PROGRAM Trips
VAR
	bTest							: BOOL;
	//delay2s : Delay2s;
	evtLogger						: FB_TcEventLogger;
	
	ACintLockRlyFaultDelay_PT		: TIME := T#2S;
	DumpRlyFaultDelay_PT			: TIME := T#2S;
	//DumpRly2FaultDelay_PT			: TIME := T#2S;
	ChrgRlyFaultDelay_PT			: TIME := T#1S;
	
	i : INT := 1;  //charger 1-8
	j : INT := 1; //section 1-3
	k : INT := 1; //section 1-4, might not need 
END_VAR


//MCP Input Trips
IF MCP_IO.MasterStopPB_Pressed = TRUE THEN
	Trips_DB.MasterStopPBPressed := TRUE;	
END_IF;

IF MCP_IO.CageEstopCircuitOK = FALSE THEN
	Trips_DB.CaseEStopCircuitBroken := TRUE; 
END_IF;

IF MCP_IO.AutoModeSelected = FALSE THEN
	Trips_DB.ManualModeSelected := TRUE; //may not be a trip
	ELSE
		Trips_DB.ManualModeSelected := FALSE;
END_IF;

IF MCP_IO.PSU1_DCOK = FALSE THEN
	Trips_DB.MCPLossDCpower := TRUE; 
END_IF;

// mapping pnumatic and dc power to trips
FOR k := 1 TO 4 BY 1 DO
	Trips_DB.Section[k].LossPneumaticPressure := LCP.Section[k].LossPneumaticPressure;
	Trips_DB.Section[k].LossDCPower := NOT LCP.Section[k].PSU1_DCOK;
END_FOR;


//any charge relay fail
IF Trips_DB.Section[1].Peak.ChargeRelay1_Failed = TRUE OR
	Trips_DB.Section[1].Peak.ChargeRelay2_Failed = TRUE OR
	Trips_DB.Section[1].Sust.ChargeRelay1_Failed = TRUE OR
	Trips_DB.Section[1].Sust.ChargeRelay2_Failed = TRUE OR
	Trips_DB.Section[2].Peak.ChargeRelay1_Failed = TRUE OR
	Trips_DB.Section[2].Peak.ChargeRelay2_Failed = TRUE OR
	Trips_DB.Section[2].Sust.ChargeRelay1_Failed = TRUE OR
	Trips_DB.Section[2].Sust.ChargeRelay2_Failed = TRUE OR
	Trips_DB.Section[3].Peak.ChargeRelay1_Failed = TRUE OR
	Trips_DB.Section[3].Peak.ChargeRelay2_Failed = TRUE OR
	Trips_DB.Section[3].Sust.ChargeRelay1_Failed = TRUE OR
	Trips_DB.Section[3].Sust.ChargeRelay2_Failed = TRUE OR
	Trips_DB.Section[4].Form.ChargeRelay1_Failed = TRUE OR 
	Trips_DB.Section[4].Form.ChargeRelay2_Failed = TRUE OR 
	Trips_DB.Section[4].Form.PreFormChrgRlyFailed = TRUE OR 
	Trips_DB.Section[4].Form.FormTrigChrgRlyFailed = TRUE OR
	Trips_DB.Section[4].Form.PreFormTrigChrgRlyFailed = TRUE		
	THEN 
		Trips_DB.AnyChargeRlyFail := TRUE;
	ELSE
		Trips_DB.AnyChargeRlyFail := FALSE;
END_IF;

//any dump relay fail
IF Trips_DB.Section[1].Peak.DumpRelay1_Failed = TRUE OR
	Trips_DB.Section[1].Peak.DumpRelay2_Failed = TRUE OR
	Trips_DB.Section[1].Sust.DumpRelay1_Failed = TRUE OR
	Trips_DB.Section[1].Sust.DumpRelay2_Failed = TRUE OR
	Trips_DB.Section[2].Peak.DumpRelay1_Failed = TRUE OR
	Trips_DB.Section[2].Peak.DumpRelay2_Failed = TRUE OR
	Trips_DB.Section[2].Sust.DumpRelay1_Failed = TRUE OR
	Trips_DB.Section[2].Sust.DumpRelay2_Failed = TRUE OR
	Trips_DB.Section[3].Peak.DumpRelay1_Failed = TRUE OR
	Trips_DB.Section[3].Peak.DumpRelay2_Failed = TRUE OR
	Trips_DB.Section[3].Sust.DumpRelay1_Failed = TRUE OR
	Trips_DB.Section[3].Sust.DumpRelay2_Failed = TRUE OR
	Trips_DB.Section[4].Form.DumpRelay1_Failed = TRUE OR 
	Trips_DB.Section[4].Form.DumpRelay2_Failed = TRUE OR 
	Trips_DB.Section[4].Form.PreFormDumpRlyFailed = TRUE OR 
	Trips_DB.Section[4].Form.FormTrigDumpRly1Failed = TRUE OR
	Trips_DB.Section[4].Form.PreFormTrigDumpRly1Failed = TRUE		
	THEN 
		Trips_DB.AnyDumpRlyFail := TRUE;
	ELSE
		Trips_DB.AnyDumpRlyFail := FALSE;
END_IF;

//if relays failed, chargers faulted, loss pneumatic pressure, or loss dc power then 
//Trips_DB.Section[j].SystemTripped := TRUE;

//system trip 
//section 1-3
FOR j := 1 TO 3 BY 1 DO
	IF Trips_DB.Section[j].LossDCPower = TRUE OR 
		Trips_DB.Section[j].LossPneumaticPressure = TRUE OR
		Trips_DB.Section[j].Peak.ChargeRelay1_Failed = TRUE OR
		Trips_DB.Section[j].Peak.ChargeRelay2_Failed = TRUE OR
		Trips_DB.Section[j].Peak.DumpRelay1_Failed = TRUE OR
		Trips_DB.Section[j].Peak.DumpRelay2_Failed = TRUE OR
		Trips_DB.Section[j].Sust.ChargeRelay1_Failed = TRUE OR
		Trips_DB.Section[j].Sust.ChargeRelay2_Failed = TRUE OR
		Trips_DB.Section[j].Sust.DumpRelay1_Failed = TRUE OR
		Trips_DB.Section[j].Sust.DumpRelay2_Failed = TRUE 
		// shorted when not supposed to ?
		THEN
			Trips_DB.Section[j].SystemTripped := TRUE;
	END_IF;
END_FOR;

//formation
IF Trips_DB.Section[4].LossDCPower = TRUE OR 
	Trips_DB.Section[4].LossPneumaticPressure = TRUE OR
	Trips_DB.Section[4].Form.ChargeRelay1_Failed = TRUE OR
	Trips_DB.Section[4].Form.ChargeRelay2_Failed = TRUE OR
	Trips_DB.Section[4].Form.DumpRelay1_Failed = TRUE OR
	Trips_DB.Section[4].Form.DumpRelay2_Failed = TRUE OR
	Trips_DB.Section[4].Form.PreFormChrgRlyFailed = TRUE OR
	Trips_DB.Section[4].Form.FormTrigChrgRlyFailed = TRUE OR
	Trips_DB.Section[4].Form.PreFormTrigChrgRlyFailed = TRUE OR
	Trips_DB.Section[4].Form.PreFormDumpRlyFailed = TRUE OR
	Trips_DB.Section[4].Form.FormTrigDumpRly1Failed = TRUE OR
	Trips_DB.Section[4].Form.PreFormTrigDumpRly1Failed = TRUE
	THEN
		Trips_DB.Section[4].SystemTripped := TRUE;
END_IF;


//Charger faults
FOR i := 1 TO 8 BY 1 DO
	//OVERTEMP 
	IF MCP_IO.Charger[i].OverTemp = TRUE THEN
		Trips_DB.AnyChargerOverTemp := TRUE;  
	END_IF;
	//Load faults
	IF MCP_IO.Charger[i].LoadFaulted = TRUE THEN
		Trips_DB.AnyChargerLoadFault := TRUE;  
	END_IF;
	//Interlock Open
	IF MCP_IO.Charger[i].InterlockOpen = TRUE THEN
		Trips_DB.AnyChargerInterlockOpen := TRUE;  
	END_IF;
	
END_FOR;

//Charger summary faults
FOR i := 1 TO 8 BY 1 DO
	IF MCP_IO.Charger[i].SummaryFaulted = TRUE THEN
		Trips_DB.AnyChargerFaulted := TRUE;  
	END_IF;
END_FOR;

//MCP trip
IF Trips_DB.AnyChargerFaulted = TRUE OR 
	Trips_DB.MasterStopPBPressed = TRUE OR
	Trips_DB.CaseEStopCircuitBroken = TRUE OR
	Trips_DB.MCPLossDCpower = TRUE 
	THEN
		Trips_DB.MCPsystemTripped := TRUE;
END_IF


//*******************E-Stop Trips
IF MCP_IO.MasterStopPB_Pressed = TRUE OR MCP_IO.CageEstopCircuitOK THEN
	Trips_DB.AnyEstopPressed := TRUE;  
END_IF;	

//*********************DC PSU
IF MCP_IO.PSU1_DCOK = TRUE AND 
	LCP.Section[1].PSU1_DCOK = TRUE AND
	LCP.Section[2].PSU1_DCOK = TRUE AND
	LCP.Section[3].PSU1_DCOK = TRUE AND
	LCP.Section[4].PSU1_DCOK = TRUE 
	THEN
		TRIPS_DB.AllDCpsuOK := TRUE;
	ELSE 
		TRIPS_DB.AllDCpsuOK := FALSE;
END_IF;

//Relay faults***************************************
//section 1 - 3
FOR j := 1 TO 3 BY 1 DO
	//Peak Charge rly1
		//fail to close
	IF LCP.Section[j].Peak.CloseChargeRelay1 = TRUE AND LCP.Section[j].Peak.ChargeRelay1_close = FALSE THEN 
		//start timer
		Trips_DB.Section[j].Peak.ChrgRly1FaultDelay_TON (IN:= TRUE, PT := ChrgRlyFaultDelay_PT);
		
		IF Trips_DB.Section[j].Peak.ChrgRly1FaultDelay_TON.Q = TRUE THEN 
			Trips_DB.Section[j].Peak.ChargeRelay1_FailtoClose := TRUE; 
			Trips_DB.Section[j].Peak.ChrgRly1FaultDelay_TON (IN:= FALSE);
		END_IF;
	ELSE
		Trips_DB.Section[j].Peak.ChrgRly1FaultDelay_TON (IN:= FALSE);
	END_IF;

		//fail to open
	IF LCP.Section[j].Peak.CloseChargeRelay1 = FALSE AND LCP.Section[j].Peak.ChargeRelay1_close = TRUE THEN 
		//start timer
		Trips_DB.Section[j].Peak.ChrgRly1FaultDelay_TON (IN:= TRUE, PT := ChrgRlyFaultDelay_PT);
		
		IF Trips_DB.Section[j].Peak.ChrgRly1FaultDelay_TON.Q = TRUE THEN 
			Trips_DB.Section[j].Peak.ChargeRelay1_FailtoOpen := TRUE; 
			Trips_DB.Section[j].Peak.ChrgRly1FaultDelay_TON (IN:= FALSE);
		END_IF;
	ELSE
		Trips_DB.Section[j].Peak.ChrgRly1FaultDelay_TON (IN:= FALSE);
	
	END_IF;

	//Peak Charge rly2	
		//fail to close
	IF LCP.Section[j].Peak.CloseChargeRelay2 = TRUE AND LCP.Section[j].Peak.ChargeRelay2_close = FALSE THEN 
		//start timer
		Trips_DB.Section[j].Peak.ChrgRly2FaultDelay_TON (IN:= TRUE, PT := ChrgRlyFaultDelay_PT);
		
		IF Trips_DB.Section[j].Peak.ChrgRly2FaultDelay_TON.Q = TRUE THEN 
			Trips_DB.Section[j].Peak.ChargeRelay2_FailtoClose := TRUE; 
			Trips_DB.Section[j].Peak.ChrgRly2FaultDelay_TON (IN:= FALSE);
		END_IF;
	ELSE
		Trips_DB.Section[j].Peak.ChrgRly2FaultDelay_TON (IN:= FALSE);
	END_IF;
	
		//fail to open
	IF LCP.Section[j].Peak.CloseChargeRelay2 = FALSE AND LCP.Section[j].Peak.ChargeRelay2_close = TRUE THEN 
		//start timer
		Trips_DB.Section[j].Peak.ChrgRly2FaultDelay_TON (IN:= TRUE, PT := ChrgRlyFaultDelay_PT);
		
		IF Trips_DB.Section[j].Peak.ChrgRly2FaultDelay_TON.Q = TRUE THEN 
			Trips_DB.Section[j].Peak.ChargeRelay2_FailtoOpen := TRUE; 
			Trips_DB.Section[j].Peak.ChrgRly2FaultDelay_TON (IN:= FALSE);
		END_IF;
	ELSE
		Trips_DB.Section[j].Peak.ChrgRly2FaultDelay_TON (IN:= FALSE);
	END_IF;

	//Peak dump rly1
		//fail to open
	IF LCP.Section[j].Peak.OpenDumpRelay1 = TRUE AND LCP.Section[j].Peak.DumpRelay1_close = TRUE THEN 
		//start timer
		Trips_DB.Section[j].Peak.DumpRly1FaultDelay_TON (IN := TRUE, PT := DumpRlyFaultDelay_PT);

		IF Trips_DB.Section[j].Peak.DumpRly1FaultDelay_TON.Q = TRUE THEN 
			Trips_DB.Section[j].Peak.DumpRelay1_FailtoOpen := TRUE; 
			Trips_DB.Section[j].Peak.DumpRly1FaultDelay_TON (IN:= FALSE);
		END_IF; 
	ELSE
		Trips_DB.Section[j].Peak.DumpRly1FaultDelay_TON (IN:= FALSE);
	END_IF;

		//fail to close
	IF LCP.Section[j].Peak.OpenDumpRelay1 = FALSE AND LCP.Section[j].Peak.DumpRelay1_close = FALSE THEN 
		//start timer
		Trips_DB.Section[j].Peak.DumpRly1FaultDelay_TON (IN := TRUE, PT := DumpRlyFaultDelay_PT); 
		
		IF Trips_DB.Section[j].Peak.DumpRly1FaultDelay_TON.Q = TRUE THEN 
			Trips_DB.Section[j].Peak.DumpRelay1_FailtoClose := TRUE;
			Trips_DB.Section[j].Peak.DumpRly1FaultDelay_TON (IN:= FALSE);
		END_IF;
	ELSE
		Trips_DB.Section[j].Peak.DumpRly1FaultDelay_TON (IN:= FALSE);
	END_IF;

	//Peak dump rly2
		//fail to open
	IF LCP.Section[j].Peak.OpenDumpRelay2 = TRUE AND LCP.Section[j].Peak.DumpRelay2_close = TRUE THEN 
		//start timer
		Trips_DB.Section[j].Peak.DumpRly2FaultDelay_TON (IN := TRUE, PT := DumpRlyFaultDelay_PT); 
		
		IF Trips_DB.Section[j].Peak.DumpRly2FaultDelay_TON.Q = TRUE THEN 
			Trips_DB.Section[j].Peak.DumpRelay2_FailtoOpen := TRUE; 
			Trips_DB.Section[j].Peak.DumpRly2FaultDelay_TON (IN:= FALSE);
		END_IF;
	ELSE
		Trips_DB.Section[j].Peak.DumpRly2FaultDelay_TON (IN:= FALSE);
	END_IF;

		//fail to close
	IF LCP.Section[j].Peak.OpenDumpRelay2 = FALSE AND LCP.Section[j].Peak.DumpRelay2_close = FALSE THEN 
		//start timer
		Trips_DB.Section[j].Peak.DumpRly2FaultDelay_TON (IN := TRUE, PT := DumpRlyFaultDelay_PT); 
		IF Trips_DB.Section[j].Peak.DumpRly2FaultDelay_TON.Q = TRUE THEN 
			Trips_DB.Section[j].Peak.DumpRelay2_FailtoClose := TRUE; 
			
		END_IF;
	ELSE
		Trips_DB.Section[j].Peak.DumpRly2FaultDelay_TON (IN:= FALSE);
	END_IF;
//*************************************************************************************************

//Sust Charge rly1
		//fail to close
	IF LCP.Section[j].Sust.CloseChargeRelay1 = TRUE AND LCP.Section[j].Sust.ChargeRelay1_close = FALSE THEN 
		//start timer
		Trips_DB.Section[j].Sust.ChrgRly1FaultDelay_TON (IN:= TRUE, PT := ChrgRlyFaultDelay_PT);
		
		IF Trips_DB.Section[j].Sust.ChrgRly1FaultDelay_TON.Q = TRUE THEN 
			Trips_DB.Section[j].Sust.ChargeRelay1_FailtoClose := TRUE; 
			Trips_DB.Section[j].Sust.ChrgRly1FaultDelay_TON (IN:= FALSE);
		END_IF;
	ELSE
		Trips_DB.Section[j].Sust.ChrgRly1FaultDelay_TON (IN:= FALSE);	
	END_IF;

		//fail to open
	IF LCP.Section[j].Sust.CloseChargeRelay1 = FALSE AND LCP.Section[j].Sust.ChargeRelay1_close = TRUE THEN 
		//start timer
		Trips_DB.Section[j].Sust.ChrgRly1FaultDelay_TON (IN:= TRUE, PT := ChrgRlyFaultDelay_PT);
		
		IF Trips_DB.Section[j].Sust.ChrgRly1FaultDelay_TON.Q = TRUE THEN 
			Trips_DB.Section[j].Sust.ChargeRelay1_FailtoOpen := TRUE; 
			Trips_DB.Section[j].Sust.ChrgRly1FaultDelay_TON (IN:= FALSE);
		END_IF;
	ELSE
		Trips_DB.Section[j].Sust.ChrgRly1FaultDelay_TON (IN:= FALSE);
	END_IF;

	//Sust Charge rly2	
		//fail to close
	IF LCP.Section[j].Sust.CloseChargeRelay2 = TRUE AND LCP.Section[j].Sust.ChargeRelay2_close = FALSE THEN 
		//start timer
		Trips_DB.Section[j].Sust.ChrgRly2FaultDelay_TON (IN:= TRUE, PT := ChrgRlyFaultDelay_PT);
		
		IF Trips_DB.Section[j].Sust.ChrgRly2FaultDelay_TON.Q = TRUE THEN 
			Trips_DB.Section[j].Sust.ChargeRelay2_FailtoClose := TRUE;
			Trips_DB.Section[j].Sust.ChrgRly2FaultDelay_TON (IN:= FALSE);
		END_IF;
	ELSE
		Trips_DB.Section[j].Sust.ChrgRly2FaultDelay_TON (IN:= FALSE);
	END_IF;
	
		//fail to open
	IF LCP.Section[j].Sust.CloseChargeRelay2 = FALSE AND LCP.Section[j].Sust.ChargeRelay2_close = TRUE THEN 
		//start timer
		Trips_DB.Section[j].Sust.ChrgRly2FaultDelay_TON (IN:= TRUE, PT := ChrgRlyFaultDelay_PT);
		
		IF Trips_DB.Section[j].Sust.ChrgRly2FaultDelay_TON.Q = TRUE THEN 
			Trips_DB.Section[j].Sust.ChargeRelay2_FailtoOpen := TRUE; 
			Trips_DB.Section[j].Sust.ChrgRly2FaultDelay_TON (IN:= FALSE);
		END_IF;
	ELSE
		Trips_DB.Section[j].Sust.ChrgRly2FaultDelay_TON (IN:= FALSE);
	END_IF;

	//Sust dump rly1
		//fail to open
	IF LCP.Section[j].Sust.OpenDumpRelay1 = TRUE AND LCP.Section[j].Sust.DumpRelay1_close = TRUE THEN 
		//start timer
		Trips_DB.Section[j].Sust.DumpRly1FaultDelay_TON (IN := TRUE, PT := DumpRlyFaultDelay_PT);

		IF Trips_DB.Section[j].Sust.DumpRly1FaultDelay_TON.Q = TRUE THEN 
			Trips_DB.Section[j].Sust.DumpRelay1_FailtoOpen := TRUE; 
			Trips_DB.Section[j].Sust.DumpRly1FaultDelay_TON (IN:= FALSE);
		END_IF; 
	ELSE
		Trips_DB.Section[j].Sust.DumpRly1FaultDelay_TON (IN:= FALSE);
	END_IF;

		//fail to close
	IF LCP.Section[j].Sust.OpenDumpRelay1 = FALSE AND LCP.Section[j].Sust.DumpRelay1_close = FALSE THEN 
		//start timer
		Trips_DB.Section[j].Sust.DumpRly1FaultDelay_TON (IN := TRUE, PT := DumpRlyFaultDelay_PT); 
		
		IF Trips_DB.Section[j].Sust.DumpRly1FaultDelay_TON.Q = TRUE THEN 
			Trips_DB.Section[j].Sust.DumpRelay1_FailtoClose := TRUE; 
			Trips_DB.Section[j].Sust.DumpRly1FaultDelay_TON (IN:= FALSE);
		END_IF;
	ELSE
		Trips_DB.Section[j].Sust.DumpRly1FaultDelay_TON (IN:= FALSE);
	END_IF;

	//Sust dump rly2
		//fail to open
	IF LCP.Section[j].Sust.OpenDumpRelay2 = TRUE AND LCP.Section[j].Sust.DumpRelay2_close = TRUE THEN 
		//start timer
		Trips_DB.Section[j].Sust.DumpRly2FaultDelay_TON (IN := TRUE, PT := DumpRlyFaultDelay_PT); 
		
		IF Trips_DB.Section[j].Sust.DumpRly2FaultDelay_TON.Q = TRUE THEN 
			Trips_DB.Section[j].Sust.DumpRelay2_FailtoOpen := TRUE; 
			Trips_DB.Section[j].Sust.DumpRly2FaultDelay_TON (IN:= FALSE);
		END_IF;
	ELSE
		Trips_DB.Section[j].Sust.DumpRly2FaultDelay_TON (IN:= FALSE);
	END_IF;

		//fail to close
	IF LCP.Section[j].Sust.OpenDumpRelay2 = FALSE AND LCP.Section[j].Sust.DumpRelay2_close = FALSE THEN 
		//start timer
		Trips_DB.Section[j].Sust.DumpRly2FaultDelay_TON (IN := TRUE, PT := DumpRlyFaultDelay_PT); 
		IF Trips_DB.Section[j].Sust.DumpRly2FaultDelay_TON.Q = TRUE THEN 
			Trips_DB.Section[j].Sust.DumpRelay2_FailtoClose := TRUE; 
			Trips_DB.Section[j].Sust.DumpRly2FaultDelay_TON (IN:= FALSE);
		END_IF;
	ELSE
		Trips_DB.Section[j].Sust.DumpRly2FaultDelay_TON (IN:= FALSE);
	END_IF;
	
END_FOR;
//****************************************	
	
//Form Charge rly1
		//fail to close
IF LCP.Section[4].Form.CloseChargeRelay1 = TRUE AND LCP.Section[4].Form.ChargeRelay1_close = FALSE THEN 
		//start timer
		Trips_DB.Section[4].Form.ChrgRly1FaultDelay_TON (IN:= TRUE, PT := ChrgRlyFaultDelay_PT);
		
		IF Trips_DB.Section[4].Form.ChrgRly1FaultDelay_TON.Q = TRUE THEN 
			Trips_DB.Section[4].Form.ChargeRelay1_FailtoClose := TRUE; 
			Trips_DB.Section[4].Form.ChrgRly1FaultDelay_TON (IN:= FALSE);
		END_IF;
	ELSE
		Trips_DB.Section[4].Form.ChrgRly1FaultDelay_TON (IN:= FALSE);		
END_IF;

		//fail to open
IF LCP.Section[4].Form.CloseChargeRelay1 = FALSE AND LCP.Section[4].Form.ChargeRelay1_close = TRUE THEN 
		//start timer
		Trips_DB.Section[4].Form.ChrgRly1FaultDelay_TON (IN:= TRUE, PT := ChrgRlyFaultDelay_PT);
		
		IF Trips_DB.Section[4].Form.ChrgRly1FaultDelay_TON.Q = TRUE THEN 
			Trips_DB.Section[4].Form.ChargeRelay1_FailtoOpen := TRUE; 
			Trips_DB.Section[4].Form.ChrgRly1FaultDelay_TON (IN:= FALSE);
		END_IF;
	ELSE
		Trips_DB.Section[4].Form.ChrgRly1FaultDelay_TON (IN:= FALSE);
END_IF;

	//Form Charge rly2	
		//fail to close
IF LCP.Section[4].Form.CloseChargeRelay2 = TRUE AND LCP.Section[4].Form.ChargeRelay2_close = FALSE THEN 
		//start timer
		Trips_DB.Section[4].Form.ChrgRly2FaultDelay_TON (IN:= TRUE, PT := ChrgRlyFaultDelay_PT);
		
		IF Trips_DB.Section[4].Form.ChrgRly2FaultDelay_TON.Q = TRUE THEN 
			Trips_DB.Section[4].Form.ChargeRelay2_FailtoClose := TRUE; 
			Trips_DB.Section[4].Form.ChrgRly2FaultDelay_TON (IN:= FALSE);
		END_IF;
	ELSE
		Trips_DB.Section[4].Form.ChrgRly2FaultDelay_TON (IN:= FALSE);
END_IF;
	
		//fail to open
IF LCP.Section[4].Form.CloseChargeRelay2 = FALSE AND LCP.Section[4].Form.ChargeRelay2_close = TRUE THEN 
		//start timer
		Trips_DB.Section[4].Form.ChrgRly2FaultDelay_TON (IN:= TRUE, PT := ChrgRlyFaultDelay_PT);
		
		IF Trips_DB.Section[4].Form.ChrgRly2FaultDelay_TON.Q = TRUE THEN 
			Trips_DB.Section[4].Form.ChargeRelay2_FailtoOpen := TRUE; 
			Trips_DB.Section[4].Form.ChrgRly2FaultDelay_TON (IN:= FALSE);
		END_IF;
	ELSE
		Trips_DB.Section[4].Form.ChrgRly2FaultDelay_TON (IN:= FALSE);
END_IF;

	//Form dump rly1
		//fail to open
IF LCP.Section[4].Form.OpenDumpRelay1 = TRUE AND LCP.Section[4].Form.DumpRelay1_close = TRUE THEN 
		//start timer
		Trips_DB.Section[4].Form.DumpRly1FaultDelay_TON (IN := TRUE, PT := DumpRlyFaultDelay_PT);

		IF Trips_DB.Section[4].Form.DumpRly1FaultDelay_TON.Q = TRUE THEN 
			Trips_DB.Section[4].Form.DumpRelay1_FailtoOpen := TRUE; 
			Trips_DB.Section[4].Form.DumpRly1FaultDelay_TON (IN:= FALSE);
		END_IF; 
	ELSE
		Trips_DB.Section[4].Form.DumpRly1FaultDelay_TON (IN:= FALSE);
END_IF;

		//fail to close
IF LCP.Section[4].Form.OpenDumpRelay1 = FALSE AND LCP.Section[4].Form.DumpRelay1_close = FALSE THEN 
		//start timer
		Trips_DB.Section[4].Form.DumpRly1FaultDelay_TON (IN := TRUE, PT := DumpRlyFaultDelay_PT); 
		
		IF Trips_DB.Section[4].Form.DumpRly1FaultDelay_TON.Q = TRUE THEN 
			Trips_DB.Section[4].Form.DumpRelay1_FailtoClose := TRUE; 
			Trips_DB.Section[4].Form.DumpRly1FaultDelay_TON (IN:= FALSE);
		END_IF;
	ELSE
		Trips_DB.Section[4].Form.DumpRly1FaultDelay_TON (IN:= FALSE);
END_IF;

	//Form dump rly2
		//fail to open
IF LCP.Section[4].Form.OpenDumpRelay2 = TRUE AND LCP.Section[4].Form.DumpRelay2_close = TRUE THEN 
		//start timer
		Trips_DB.Section[4].Form.DumpRly2FaultDelay_TON (IN := TRUE, PT := DumpRlyFaultDelay_PT); 
		
		IF Trips_DB.Section[4].Form.DumpRly2FaultDelay_TON.Q = TRUE THEN 
			Trips_DB.Section[4].Form.DumpRelay2_FailtoOpen := TRUE; 
			Trips_DB.Section[4].Form.DumpRly2FaultDelay_TON (IN:= FALSE);
		END_IF;
	ELSE
		Trips_DB.Section[4].Form.DumpRly2FaultDelay_TON (IN:= FALSE);
END_IF;

		//fail to close
IF LCP.Section[4].Form.OpenDumpRelay2 = FALSE AND LCP.Section[4].Form.DumpRelay2_close = FALSE THEN 
		//start timer
		Trips_DB.Section[4].Form.DumpRly2FaultDelay_TON (IN := TRUE, PT := DumpRlyFaultDelay_PT); 
		IF Trips_DB.Section[4].Form.DumpRly2FaultDelay_TON.Q = TRUE THEN 
			Trips_DB.Section[4].Form.DumpRelay2_FailtoClose := TRUE; 
			Trips_DB.Section[4].Form.DumpRly2FaultDelay_TON (IN:= FALSE);
		END_IF;
	ELSE
		Trips_DB.Section[4].Form.DumpRly2FaultDelay_TON (IN:= FALSE);
END_IF;	

	//PreForm Charge rly
		//fail to close
IF (LCP.Section[4].Form.ClosePreFormChargeRly = TRUE AND LCP.Section[4].Form.PreFormChargeRly_close = FALSE) OR 
		(LCP.Section[4].Form.ClosePreFormChargeRly = FALSE AND LCP.Section[4].Form.PreFormChargeRly_close = TRUE) 
		THEN 
		//start timer
		Trips_DB.Section[4].Form.PreFormChrgRlyFaultDelay_TON (IN:= TRUE, PT := ChrgRlyFaultDelay_PT);
		
		IF Trips_DB.Section[4].Form.PreFormChrgRlyFaultDelay_TON.Q = TRUE THEN 
			Trips_DB.Section[4].Form.PreFormChrgRlyFailed := TRUE; 
			Trips_DB.Section[4].Form.PreFormChrgRlyFaultDelay_TON (IN:= FALSE);
		END_IF;
	ELSE
		Trips_DB.Section[4].Form.PreFormChrgRlyFaultDelay_TON (IN:= FALSE);
END_IF;

//form trigger charge 
		//fail to close
IF (LCP.Section[4].Form.CloseFormTrigChargeRly = TRUE AND LCP.Section[4].Form.FormTrigChargeRly_close = FALSE) OR 
		(LCP.Section[4].Form.CloseFormTrigChargeRly = FALSE AND LCP.Section[4].Form.FormTrigChargeRly_close = TRUE) 
		THEN 
		//start timer
		Trips_DB.Section[4].Form.FormTrigChrgRlyFaultDelay_TON (IN:= TRUE, PT := ChrgRlyFaultDelay_PT);
		
		IF Trips_DB.Section[4].Form.FormTrigChrgRlyFaultDelay_TON.Q = TRUE THEN 
			Trips_DB.Section[4].Form.FormTrigChrgRlyFailed := TRUE; 
			Trips_DB.Section[4].Form.FormTrigChrgRlyFaultDelay_TON (IN:= FALSE);
		END_IF;
	ELSE
		Trips_DB.Section[4].Form.FormTrigChrgRlyFaultDelay_TON (IN:= FALSE);
END_IF;

//preform trigger charge
		//fail to close
IF (LCP.Section[4].Form.ClosePreFormTrigChargeRly = TRUE AND LCP.Section[4].Form.PreFormTrigChargeRly_close = FALSE) OR 
		(LCP.Section[4].Form.ClosePreFormTrigChargeRly = FALSE AND LCP.Section[4].Form.PreFormTrigChargeRly_close = TRUE) 
		THEN 
		//start timer
		Trips_DB.Section[4].Form.PreFormTrigChrgRlyFaultDelay_TON (IN:= TRUE, PT := ChrgRlyFaultDelay_PT);
		
		IF Trips_DB.Section[4].Form.PreFormTrigChrgRlyFaultDelay_TON.Q = TRUE THEN 
			Trips_DB.Section[4].Form.PreFormTrigChrgRlyFailed := TRUE; 
			Trips_DB.Section[4].Form.PreFormTrigChrgRlyFaultDelay_TON (IN:= FALSE);
		END_IF;
	ELSE
		Trips_DB.Section[4].Form.PreFormTrigChrgRlyFaultDelay_TON (IN:= FALSE);
END_IF;

//preform dump
	//fail to close
IF (LCP.Section[4].Form.OpenPreFormDumpRly = TRUE AND LCP.Section[4].Form.PreFormDumpRly_close = FALSE) OR 
		(LCP.Section[4].Form.OpenPreFormDumpRly = FALSE AND LCP.Section[4].Form.PreFormDumpRly_close = TRUE) 
		THEN 
		//start timer
		Trips_DB.Section[4].Form.PreFormDumpRlyFaultDelay_TON (IN:= TRUE, PT := DumpRlyFaultDelay_PT);
		
		IF Trips_DB.Section[4].Form.PreFormDumpRlyFaultDelay_TON.Q = TRUE THEN 
			Trips_DB.Section[4].Form.PreFormDumpRlyFailed := TRUE; 
			Trips_DB.Section[4].Form.PreFormDumpRlyFaultDelay_TON (IN:= FALSE);
		END_IF;
	ELSE
		Trips_DB.Section[4].Form.PreFormDumpRlyFaultDelay_TON (IN:= FALSE);
END_IF;

//form trigger dump
	//fail to close
IF (LCP.Section[4].Form.OpenFormTrigDumpRly1 = TRUE AND LCP.Section[4].Form.FormTrigDumpRly1_close = FALSE) OR 
		(LCP.Section[4].Form.OpenFormTrigDumpRly1 = FALSE AND LCP.Section[4].Form.FormTrigDumpRly1_close = TRUE) 
		THEN 
		//start timer
		Trips_DB.Section[4].Form.FormTrigDumpRlyFaultDelay_TON (IN:= TRUE, PT := DumpRlyFaultDelay_PT);
		
		IF Trips_DB.Section[4].Form.FormTrigDumpRlyFaultDelay_TON.Q = TRUE THEN 
			Trips_DB.Section[4].Form.FormTrigDumpRly1Failed := TRUE; 
			Trips_DB.Section[4].Form.FormTrigDumpRlyFaultDelay_TON (IN:= FALSE);
		END_IF;
	ELSE
		Trips_DB.Section[4].Form.FormTrigDumpRlyFaultDelay_TON (IN:= FALSE);
END_IF;
	
//preform trigger dump
	//fail to close
IF (LCP.Section[4].Form.OpenPreFormTrigDumpRly1 = TRUE AND LCP.Section[4].Form.PreFormTrigDumpRly1_close = FALSE) OR 
		(LCP.Section[4].Form.OpenPreFormTrigDumpRly1 = FALSE AND LCP.Section[4].Form.PreFormTrigDumpRly1_close = TRUE) 
		THEN 
		//start timer
		Trips_DB.Section[4].Form.PreFormTrigDumpRlyFaultDelay_TON (IN:= TRUE, PT := DumpRlyFaultDelay_PT);
		
		IF Trips_DB.Section[4].Form.PreFormTrigDumpRlyFaultDelay_TON.Q = TRUE THEN 
			Trips_DB.Section[4].Form.PreFormTrigDumpRly1Failed := TRUE; 
			Trips_DB.Section[4].Form.PreFormTrigDumpRlyFaultDelay_TON (IN:= FALSE);
		END_IF;
	ELSE
		Trips_DB.Section[4].Form.PreFormTrigDumpRlyFaultDelay_TON (IN:= FALSE);
END_IF;
	

// if rly fail to close or fail to open then trips_db.rly_failed - for alarms	
FOR j := 1 TO 3 BY 1 DO
	//peak
	IF Trips_DB.Section[j].Peak.ChargeRelay1_FailtoClose = TRUE OR Trips_DB.Section[j].Peak.ChargeRelay1_FailtoOpen = TRUE THEN
		Trips_DB.Section[j].Peak.ChargeRelay1_Failed := TRUE;  
	END_IF;
	
	IF Trips_DB.Section[j].Peak.ChargeRelay2_FailtoClose = TRUE OR Trips_DB.Section[j].Peak.ChargeRelay2_FailtoOpen = TRUE THEN
		Trips_DB.Section[j].Peak.ChargeRelay2_Failed := TRUE;  
	END_IF;
	
	IF Trips_DB.Section[j].Peak.DumpRelay1_FailtoClose = TRUE OR Trips_DB.Section[j].Peak.DumpRelay1_FailtoOpen = TRUE THEN
		Trips_DB.Section[j].Peak.DumpRelay1_Failed := TRUE;  
	END_IF;
	
	IF Trips_DB.Section[j].Peak.DumpRelay2_FailtoClose = TRUE OR Trips_DB.Section[j].Peak.DumpRelay2_FailtoOpen = TRUE THEN
		Trips_DB.Section[j].Peak.DumpRelay2_Failed := TRUE;  
	END_IF;
	
	//sust
	IF Trips_DB.Section[j].Sust.ChargeRelay1_FailtoClose = TRUE OR Trips_DB.Section[j].Sust.ChargeRelay1_FailtoOpen = TRUE THEN
		Trips_DB.Section[j].Sust.ChargeRelay1_Failed := TRUE;  
	END_IF;
	
	IF Trips_DB.Section[j].Sust.ChargeRelay2_FailtoClose = TRUE OR Trips_DB.Section[j].Sust.ChargeRelay2_FailtoOpen = TRUE THEN
		Trips_DB.Section[j].Sust.ChargeRelay2_Failed := TRUE;  
	END_IF;
	
	IF Trips_DB.Section[j].Sust.DumpRelay1_FailtoClose = TRUE OR Trips_DB.Section[j].Sust.DumpRelay1_FailtoOpen = TRUE THEN
		Trips_DB.Section[j].Sust.DumpRelay1_Failed := TRUE;  
	END_IF;
	
	IF Trips_DB.Section[j].Sust.DumpRelay2_FailtoClose = TRUE OR Trips_DB.Section[j].Sust.DumpRelay2_FailtoOpen = TRUE THEN
		Trips_DB.Section[j].Sust.DumpRelay2_Failed := TRUE;  
	END_IF;
	
END_FOR;

// no faulted detected
IF Trips_DB.MCPsystemTripped = FALSE AND
	Trips_DB.AnyChargerOverTemp = FALSE AND
	Trips_DB.AnyChargerLoadFault = FALSE AND
	Trips_DB.AnyChargerInterlockOpen = FALSE AND
	Trips_DB.AnyChargerFaulted = FALSE AND
	Trips_DB.AnyEstopPressed = FALSE AND
	Trips_DB.AnyDumpRlyFail = FALSE AND
	Trips_DB.AnyChargeRlyFail = FALSE
	THEN
		Trips_DB.NoFaultDetected := TRUE;
	ELSE
		Trips_DB.NoFaultDetected := FALSE;
END_IF;


(*
FOR i := 1 TO 10 BY 1 DO
	IF (Trips_DB.Coil[i].ACInterlockRelayFailedtoClose = TRUE OR 
		Trips_DB.Coil[i].ACInterlockRelayFailedtoOpen = TRUE OR 
		Trips_DB.Coil[i].ChargeRelay_FailtoClose = TRUE OR
		Trips_DB.Coil[i].ChargeRelay_FailtoOpen = TRUE OR
		Trips_DB.Coil[i].DumpRelay1_FailtoClose =  TRUE OR 
		Trips_DB.Coil[i].DumpRelay1_FailtoOpen = TRUE OR 
		Trips_DB.Coil[i].DumpRelay2_FailtoClose =  TRUE OR 
		Trips_DB.Coil[i].DumpRelay2_FailtoOpen = TRUE OR 
		Trips_DB.Coil[i].ChargerVoltageReadingFaulted = TRUE OR
		Trips_DB.Coil[i].CurrentReadingFaulted = TRUE OR
		Devices.Coil[i].Local_EstopPB_Pressed = TRUE OR
		Devices.Coil[i].LossPneumaticPressure = FALSE) AND Devices.Coil[i].CoilEnabled = TRUE 	
		THEN
			Devices.Coil[i].SystemFaulted := TRUE;
	END_IF
	
	IF Devices.Coil[i].SystemFaulted = TRUE THEN
		Trips_DB.SystemTripped := TRUE;
	END_IF;
END_FOR;

//*********************************** Test
(*IF InstrumentReading.R2_01_CH01 <= 0.0 THEN
	delay2s(input := FALSE);
ELSE 
	delay2s (input := TRUE);
END_IF;
bTest := delay2s.output;
*)
// Instrumentation Hardware trip
//Input.R2_01_00_Status.0;
*)
//************** Clear System Fault
IF Trips_DB.ClearAllFaults THEN
	//Trips_DB.InstrumentationFaulted := FALSE;
	//Trips_DB.SystemTripped := FALSE;
	Trips_DB.MCPsystemTripped := FALSE; //reset mcp trip
	Trips_DB.AnyChargerOverTemp := FALSE;
	Trips_DB.AnyChargerLoadFault := FALSE;  
	Trips_DB.AnyChargerInterlockOpen := FALSE;
	Trips_DB.AnyChargerFaulted := FALSE;
	Trips_DB.AnyEstopPressed := FALSE;
	Trips_DB.AnyDumpRlyFail := FALSE;
	Trips_DB.AnyChargeRlyFail := FALSE;
	Trips_DB.MasterStopPBPressed := FALSE; //this is only for alarms
	Trips_DB.CaseEStopCircuitBroken := FALSE;
	Trips_DB.MCPLossDCpower := FALSE;
	//Trips_DB.AnyACInterlockFail := FALSE;
	//reset relay trips
	FOR j := 1 TO 3 BY 1 DO 
		//reset relay faults
		Trips_DB.Section[j].SystemTripped := FALSE;
		//Peaking
		Trips_DB.Section[j].Peak.DumpRelay1_FailtoClose := FALSE;
		Trips_DB.Section[j].Peak.DumpRelay1_FailtoOpen := FALSE;
		Trips_DB.Section[j].Peak.DumpRelay2_FailtoClose := FALSE;
		Trips_DB.Section[j].Peak.DumpRelay2_FailtoOpen := FALSE;
		Trips_DB.Section[j].Peak.ChargeRelay1_FailtoClose := FALSE;
		Trips_DB.Section[j].Peak.ChargeRelay1_FailtoOpen := FALSE;
		Trips_DB.Section[j].Peak.ChargeRelay2_FailtoClose := FALSE;
		Trips_DB.Section[j].Peak.ChargeRelay2_FailtoOpen := FALSE;
		//Sust
		Trips_DB.Section[j].Sust.DumpRelay1_FailtoClose := FALSE;
		Trips_DB.Section[j].Sust.DumpRelay1_FailtoOpen := FALSE;
		Trips_DB.Section[j].Sust.DumpRelay2_FailtoClose := FALSE;
		Trips_DB.Section[j].Sust.DumpRelay2_FailtoOpen := FALSE;
		Trips_DB.Section[j].Sust.ChargeRelay1_FailtoClose := FALSE;
		Trips_DB.Section[j].Sust.ChargeRelay1_FailtoOpen := FALSE;
		Trips_DB.Section[j].Sust.ChargeRelay2_FailtoClose := FALSE;
		Trips_DB.Section[j].Sust.ChargeRelay2_FailtoOpen := FALSE;
	
	END_FOR;
	
	//FORM
	Trips_DB.Section[4].Form.ChargeRelay1_FailtoOpen := FALSE;
	Trips_DB.Section[4].Form.ChargeRelay1_FailtoClose := FALSE;
	Trips_DB.Section[4].Form.ChargeRelay1_Failed:= FALSE;
	Trips_DB.Section[4].Form.ChargeRelay2_FailtoOpen := FALSE;
	Trips_DB.Section[4].Form.ChargeRelay2_FailtoClose := FALSE;
	Trips_DB.Section[4].Form.ChargeRelay2_Failed:= FALSE;
	
	Trips_DB.Section[4].Form.DumpRelay1_FailtoOpen := FALSE;
	Trips_DB.Section[4].Form.DumpRelay1_FailtoClose := FALSE;
	Trips_DB.Section[4].Form.DumpRelay1_Failed := FALSE;
	Trips_DB.Section[4].Form.DumpRelay2_FailtoOpen := FALSE;
	Trips_DB.Section[4].Form.DumpRelay2_FailtoClose := FALSE;
	Trips_DB.Section[4].Form.DumpRelay2_Failed := FALSE;
	
	Trips_DB.Section[4].Form.PreFormChrgRlyFailed := FALSE;
	Trips_DB.Section[4].Form.FormTrigChrgRlyFailed := FALSE;
	Trips_DB.Section[4].Form.PreFormTrigChrgRlyFailed := FALSE;
	Trips_DB.Section[4].Form.PreFormDumpRlyFailed := FALSE;
	Trips_DB.Section[4].Form.FormTrigDumpRly1Failed := FALSE;
	Trips_DB.Section[4].Form.PreFormTrigDumpRly1Failed := FALSE;
	
	Trips_DB.Section[4].SystemTripped := FALSE;
	
	evtLogger.ClearAllAlarms(0, FALSE);
	//evtLogger.ClearLoggedEvents(1);
END_IF;


IF i > 8 THEN 
	i := 1;
END_IF;

IF j > 3 THEN 
	j := 1;
END_IF;

IF k > 4 THEN 
	k := 1;
END_IF;

END_PROGRAM

(* stored: Version 1.1.0.1, ProductVersion 3.1.4024.11
   POU Trips: Id {4df83c48-b93a-45f7-abb7-3e8fd700423f}, SpecialFunc None *)
